// TIA Portal V20 export
TYPE "typeEm0Commands"
// stored: Access Published, Namespace Unit1
   STRUCT
      jobinterface { ExternalWritable := 'False'} : "Unit1.typeEm0CommandsJobInterface";
   END_STRUCT;
END_TYPE
